TYPE ST_APP_STATE :
STRUCT
  AppInit             : E_PROGRESS;
  AppState            : E_INSTANCE_STATE;
END_STRUCT
END_TYPE

(* stored: Version 1.1.0.1, ProductVersion 3.1.4026.13
   DUT ST_APP_STATE: Id {8ad5dcc9-9492-4d8e-972f-a2d6ca9938d0} *)
